(* Copyright (c) 2015 Fausto Bellei - fbellei@creoevolution.com - CREO EVOLUTION SRL - http://www.creoevolution.com *)

(* Permission is hereby granted, free of charge, to any person obtaining a copy of this software and associated documentation files (the "Software"), to deal in the
   Software without restriction, including without limitation the rights to use, copy, modify, merge, publish, distribute, sublicense, and/or sell copies of the Software,
   and to permit persons to whom the Software is furnished to do so, subject to the following conditions:

   The above copyright notice and this permission notice shall be included in all copies or substantial portions of the Software.

   THE SOFTWARE IS PROVIDED "AS IS", WITHOUT WARRANTY OF ANY KIND, EXPRESS OR IMPLIED, INCLUDING BUT NOT LIMITED TO THE WARRANTIES OF
   MERCHANTABILITY, FITNESS FOR A PARTICULAR PURPOSE AND NONINFRINGEMENT. IN NO EVENT SHALL THE AUTHORS OR COPYRIGHT HOLDERS BE LIABLE FOR
   ANY CLAIM, DAMAGES OR OTHER LIABILITY, WHETHER IN AN ACTION OF CONTRACT, TORT OR OTHERWISE, ARISING FROM, OUT OF OR IN CONNECTION WITH THE
   SOFTWARE OR THE USE OR OTHER DEALINGS IN THE SOFTWARE. *)

FUNCTION_BLOCK TFGateAccessDoppiaMacchina
VAR_INPUT
	MachineCmd : POINTER TO CommandBuffer;
	MachineCmdExe : POINTER TO CommandExe;
	MachineState : POINTER TO State;
	MachineError : POINTER TO Error;
	MachineMode : POINTER TO Mode;
	
	MachineCmd2 : POINTER TO CommandBuffer;//Macchina 2
	MachineCmdExe2 : POINTER TO CommandExe;//Macchina 2
	MachineState2 : POINTER TO State;//Macchina 2
	MachineError2 : POINTER TO Error;//Macchina 2
	MachineMode2 : POINTER TO Mode;//Macchina 2

	TimeBase : REAL;
	AccessRequest : BOOL;
	AccessDone : BOOL;
	LGVAccessActive	: BOOL;
	TilterPhaseStopDone : BOOL;
	PowerOK : BOOL;//Indica la presenza della marcia
END_VAR
VAR_OUTPUT
	AccessLamp : BOOL; (* Access Lamp: 	OFF = No Access Consent,
										ON = Access Consent,
										FLASH (1sec) = Access Requested (Machine Stopping)
										FLASH (0.5sec) = Waiting Restart
										FLASH (0.1sec) = Access Error *)
										
	AccesActive : BOOL; (* Gate Acces Sequence in Execution *)
	AccessOK : BOOL;	(* Accesso consentito *)
	TilterPhaseStop : BOOL;		
	AccessERRORCode : UINT;		
	ErrAck : BOOL;
	ErrAckDriver : BOOL;			
END_VAR
VAR
	ParametersArray : ParametersArray;
	
	AccessERROR : BOOL;
	AccessReqIN : BOOL;
	AccessReqOUT : BOOL;
	AccessCase : INT;
	MachineWasRunning : BOOL;
	MachineWasRunning2 : bool;
	Timer100 : REAL;
	Timer500 : REAL;
	Timer1000 : REAL;
	Clock100 : BOOL;
	Clock500 : BOOL;
	Clock1000 : BOOL;
	TimerPowerOFF : real;
	MEMDiMarciaInPartenza : BOOL;
	TimerRitardoPower : REAL;
END_VAR

TFTimerCall(ADR(Timer100),TimeBase);
TFTimerCall(ADR(Timer500),TimeBase);
TFTimerCall(ADR(Timer1000),TimeBase);
TFTimerCall(ADR(TimerPowerOFF),TimeBase);
TFTimerCall(ADR(TimerRitardoPower),TimeBase);

CASE AccessCase OF
	
	(* Wait Request ON *)
	0:	AccesActive := FALSE;
		AccessOK := FALSE;
		AccessReqIN := FALSE;
		AccessReqOUT := FALSE;
		
		IF AccessRequest AND NOT AccessDone (*AND NOT LGVAccessActive*) AND NOT TFIsModuleError(MachineError^) AND NOT TFIsModuleError(MachineError2^) THEN
			AccesActive := TRUE;
			AccessERROR := FALSE;
			AccessReqIN := TRUE;
			(* Machine Was Running if CmdDO and No Stop Request *) 
			MachineWasRunning := MachineCmdExe^.Code = CmdDO AND MachineCmdExe^.PhaseStopRequest = 0 AND MachineCmdExe^.RapidStopRequest = 0;
			MachineWasRunning2 := MachineCmdExe2^.Code = CmdDO AND MachineCmdExe2^.PhaseStopRequest = 0 AND MachineCmdExe2^.RapidStopRequest = 0;
			AccessCase := 10;
		ELSIF AccessERROR THEN
			AccessERRORCode := 0;
			AccessERROR := FALSE;
			TilterPhaseStop := false;
		END_IF
		
	(* Phase Stop *)
	10:	TFParametersArrayClear(ADR(ParametersArray));
		TFCommandSend(CmdSTOPPHASE,ParametersArray,MachineCmd^);
		TFCommandSend(CmdSTOPPHASE,ParametersArray,MachineCmd2^);
		AccessCase := AccessCase + 1;
		
	11:	IF ((TFStateCodeGet(MachineState^) = StateDO_END OR
			MachineCmdExe^.Code = CmdNOP)) AND
			((TFStateCodeGet(MachineState2^) = StateDO_END OR
			MachineCmdExe2^.Code = CmdNOP)) THEN
				TFTimerSet(ADR(TimerPowerOFF),100,TRUE);
				AccessCase := 20;
		ELSIF TFIsModuleError(MachineError^) OR TFIsModuleError(MachineError2^) THEN
			AccessERRORCode := ErrMACHINEPALLETIZER_ERRORE_MACCHINA_IN_RICHIN;
			TilterPhaseStop := TRUE;
			AccessERROR := TRUE;
			AccessCase := 0;
		END_IF

	(* Power Off *)
	20:	//Valuto se nel pal è presente la marcia, in questo modo alla fine della rich. di ingresso do o meno il power
		IF PowerOK THEN
			MEMDiMarciaInPartenza := TRUE;
		ELSE
			MEMDiMarciaInPartenza := FALSE;
		END_IF
		IF TFTimerDone(ADR(TimerPowerOFF)) THEN
			TilterPhaseStop := FALSE;
			TFParametersArrayClear(ADR(ParametersArray));
			ParametersArray.Parameters[0] := '0';
			TFCommandSend(CmdPOWER,ParametersArray,MachineCmd^);
			TFCommandSend(CmdPOWER,ParametersArray,MachineCmd2^);
			AccessCase := AccessCase + 1;
		ELSIF TFIsModuleError(MachineError^) OR  TFIsModuleError(MachineError2^) THEN
			AccessERRORCode := ErrMACHINEPALLETIZER_ERRORE_MACCHINA_IN_RICHIN;
			AccessERROR := TRUE;
			AccessCase := 0;
		ELSIF NOT AccessRequest THEN
			TilterPhaseStop := FALSE;
			AccessCase := 0;
		END_IF	

	21:	IF TFStateCodeGet(MachineState^) = StatePOWER_END AND TFStateCodeGet(MachineState2^) = StatePOWER_END THEN
			AccessCase := 25;
		ELSIF TFIsModuleError(MachineError^) OR TFIsModuleError(MachineError2^) THEN
			AccessERRORCode := ErrMACHINEPALLETIZER_ERRORE_MACCHINA_IN_RICHIN;
			AccessERROR := TRUE;
			AccessCase := 0;
		END_IF
		
	25:(* Access Ok.... Wait Request Done ON *)
		AccessReqIN := FALSE;
		AccessReqOUT := FALSE;
		AccessOK := TRUE;
		IF NOT AccessRequest AND AccessDone THEN
			AccessCase := AccessCase + 1;
			TFTimerSet(ADR(TimerRitardoPower),100,TRUE);
			ErrAck := TRUE;
		END_IF
		IF TFIsModuleError(MachineError^) OR TFIsModuleError(MachineError2^) THEN
			AccessERRORCode := ErrMACHINEPALLETIZER_ERRORE_MACCHINA_IN_RICHIN;
			AccessERROR := TRUE;
			AccessCase := 0;
		END_IF
		
	26:
		IF TFTimerDone(ADR(TimerRitardoPower)) THEN
			TFTimerSet(ADR(TimerRitardoPower),100,TRUE);
			ErrAck := FALSE;
			AccessCase := 27;
		END_IF
		
	27:
		IF TFTimerDone(ADR(TimerRitardoPower)) THEN
			TFTimerSet(ADR(TimerRitardoPower),100,TRUE);
			ErrAckDriver := TRUE;
			AccessCase := 30;
		END_IF

	(* Access Ok.... Wait Request Done ON *)
	30:	//AccessReqIN := FALSE;
		//AccessReqOUT := FALSE;
		//AccessOK := TRUE;
		//IF NOT AccessRequest AND AccessDone THEN
		IF TFTimerDone(ADR(TimerRitardoPower)) THEN
			AccessCase := 31;
			TFTimerSet(ADR(TimerRitardoPower),100,TRUE);
			ErrAckDriver := FALSE;
		END_IF
		//END_IF
		IF TFIsModuleError(MachineError^) OR TFIsModuleError(MachineError2^) THEN
			AccessERRORCode := ErrMACHINEPALLETIZER_ERRORE_MACCHINA_IN_RICHIN;
			AccessERROR := TRUE;
			AccessCase := 0;
		END_IF

	(* Wait Request Done OFF *)
	31:	TFTimerSet(ADR(TimerRitardoPower),100,AccessDone);
		IF NOT AccessDone AND TFTimerDone(ADR(TimerRitardoPower))THEN
			AccessOK := FALSE;
			AccessReqOUT := TRUE;
			AccessCase := 40;
			ErrAckDriver := FALSE;
		ELSIF TFIsModuleError(MachineError^) OR TFIsModuleError(MachineError2^) THEN
			AccessERRORCode := ErrMACHINEPALLETIZER_ERRORE_MACCHINA_IN_RICHIN;
			AccessERROR := TRUE;
			AccessCase := 0;
		END_IF
		
	(* Power ON *)
	40:	IF NOT LGVAccessActive THEN
			IF MEMDiMarciaInPartenza THEN
				TFParametersArrayClear(ADR(ParametersArray));
				ParametersArray.Parameters[0] := '1';
				TFCommandSend(CmdPOWER,ParametersArray,MachineCmd^);
				TFCommandSend(CmdPOWER,ParametersArray,MachineCmd2^);
				AccessCase := AccessCase + 1;
			ELSE
				AccessCase := 50;
			END_IF		
		ELSE
			AccessCase := 50;
		END_IF	

	41:	IF TFStateCodeGet(MachineState^) = StatePOWER_END AND  TFStateCodeGet(MachineState2^) = StatePOWER_END THEN //OR TFIsModuleError(MachineError^) THEN
			AccessCase := 50;
		ELSIF TFIsModuleError(MachineError^) OR TFIsModuleError(MachineError2^) THEN
			AccessERRORCode := ErrMACHINEPALLETIZER_ERRORE_MACCHINA_IN_RICHIN;
			AccessERROR := TRUE;
			AccessCase := 0;
		END_IF

	50:	IF NOT AccessRequest AND AccessDone THEN
			AccessCase := AccessCase + 1;
		END_IF

	(* Wait Request Done OFF *)
	51:	IF NOT AccessDone THEN
			AccessCase := 60;
		END_IF

	(* Machine Restart *)
	60:	AccessCase := AccessCase + 1;
		IF MachineWasRunning AND
			MachineMode^.Auto AND
			NOT MachineMode^.StopRequest AND
			NOT MachineMode^.RapidStopRequest AND NOT LGVAccessActive THEN
				TFParametersArrayClear(ADR(ParametersArray));
				TFCommandSend(CmdDO,ParametersArray,MachineCmd^);		
		ELSIF TFIsModuleError(MachineError^) THEN
			AccessERRORCode := ErrMACHINEPALLETIZER_ERRORE_MACCHINA_IN_RICHIN;
			AccessERROR := TRUE;
			AccessCase := 0;
		END_IF
		IF MachineWasRunning2 AND
			MachineMode2^.Auto AND
			NOT MachineMode2^.StopRequest AND
			NOT MachineMode2^.RapidStopRequest AND NOT LGVAccessActive THEN
				TFParametersArrayClear(ADR(ParametersArray));
				TFCommandSend(CmdDO,ParametersArray,MachineCmd2^);		
		ELSIF TFIsModuleError(MachineError2^) THEN
			AccessERRORCode := ErrMACHINEPALLETIZER_ERRORE_MACCHINA_IN_RICHIN;
			AccessERROR := TRUE;
			AccessCase := 0;
		END_IF
			
	61:	AccessReqIN := FALSE;
		AccessReqOUT := FALSE;
		AccessOK := FALSE;
		AccessCase := 0;
		MEMDiMarciaInPartenza := FALSE;
		
	ELSE
		AccessERROR := TRUE;
		AccessERRORCode := ErrMACHINEPALLETIZER_ERRORE_MACCHINA_IN_RICHIN;
		MEMDiMarciaInPartenza := FALSE;
		AccessCase := 0;
		
END_CASE

(* Clocks *)
IF TFTimerDone(ADR(Timer100)) THEN
	TFTimerSet(ADR(Timer100),100,TRUE);
	Clock100 := NOT Clock100;
END_IF
IF TFTimerDone(ADR(Timer500)) THEN
	TFTimerSet(ADR(Timer500),500,TRUE);
	Clock500 := NOT Clock500;
END_IF
IF TFTimerDone(ADR(Timer1000)) THEN
	TFTimerSet(ADR(Timer1000),1000,TRUE);
	Clock1000 := NOT Clock1000;
END_IF

(* Access Lamp *)
AccessLamp := 	(AccessOK OR
				(AccessReqOUT AND Clock500) OR
				(AccessReqIN AND Clock1000))AND
				NOT AccessERROR OR (AccessERROR AND Clock100);

END_FUNCTION_BLOCK

(* stored: Version 1.1.0.1, ProductVersion 3.1.4024.11
   POU TFGateAccessDoppiaMacchina: Id {8d7af665-1c33-4df7-b8ca-b623c061c337}, SpecialFunc None *)
